FUNCTION_BLOCK Test_IteratorReturnsTests EXTENDS T_UnitTestBase
VAR
    List     : T_ListOfTests(Capacity := 10);
    Iterator : T_TestIterator;
    Test0 : Test_ExampleTest(0);
    Test1 : Test_ExampleTest(0);
    Test2 : Test_ExampleTest(0);
    Test3 : Test_ExampleTest(0);
END_VAR

METHOD Init
List.Clear();

List.AddTest(Test0);
List.AddTest(Test1);
List.AddTest(Test2);
List.AddTest(Test3);
END_METHOD

PROPERTY Name : Tc2_System.T_MaxString
GET
END_GET
END_PROPERTY

METHOD RunTest
VAR_OUTPUT
    TestCompleted : BOOL;
    TestFailed    : BOOL;
END_VAR
VAR_INST
    Test2_InterfacePointer : I_UnitTest;
    ReturnValue            : I_UnitTest;
END_VAR
Iterator.Initialise(List);
Iterator.GetNext();
Iterator.GetNext();

Test2_InterfacePointer := Test2;
ReturnValue            := Iterator.GetNext();

AssertEquals(Source   := TestName,
               Expected := Test2_InterfacePointer,
               Actual   := ReturnValue,
               Message  := 'Interface pointer TestNumber2 was not correct',
               Failed   => TestFailed);

TestCompleted := TRUE;
END_METHOD

END_FUNCTION_BLOCK

(* stored: Version 1.1.0.1, ProductVersion 3.1.4024.12
   POU Test_IteratorReturnsTests: Id {85ba2117-52d5-4804-a1bf-0980042b7edf}, SpecialFunc None
   Method Init: Id {f5cf7b1f-1614-4f76-ad11-f946fcc59d0a}
   Property Name: Id {61ffc133-d5b1-40ed-ba9f-c11825891419}
   Get Get: Id {80eafa1c-22c1-4ceb-8368-382c827b6458}
   Method RunTest: Id {ad0316aa-803b-48e0-9d3d-7922c261ce32} *)
